FUNCTION_BLOCK Simulation
VAR_INPUT
END_VAR
VAR_OUTPUT
END_VAR
VAR
	tonTaktgeber: ton;	

	xAuslass1: BOOL;	//Es wird Wasser abgelassen
	xAuslass2: BOOL;
	xAuslass3: BOOL;

	uiFuellstandTank1: UINT;	// 0 --> voll; 300 --> leer
	uiFuellstandTank2: UINT;
	uiFuellstandTank3: UINT;	
END_VAR

//Simulation für die Visualisierung
tonTaktgeber(IN:= NOT tonTaktgeber.Q, PT:= T#30MS);

IF tonTaktgeber.Q THEN
	// damit das Simulation mit passabler Geschwindigkeit läuft	

	// Tank leeren
	IF  xAuslass1 THEN
		IF uiFuellstandTank1 < 300 THEN
			uiFuellstandTank1 := uiFuellstandTank1 + 1;
		ELSE
			uiFuellstandTank1 := 300;		
		END_IF
	END_IF

	IF  xAuslass2 THEN
		IF uiFuellstandTank2 < 300 THEN
			uiFuellstandTank2 := uiFuellstandTank2 + 1;
		ELSE
			uiFuellstandTank2 := 300;		
		END_IF
	END_IF

	IF  xAuslass3 THEN
		IF uiFuellstandTank3 < 300 THEN
			uiFuellstandTank3 := uiFuellstandTank3 + 1;
		ELSE
			uiFuellstandTank3 := 300;		
		END_IF
	END_IF
	
	// Tank füllen
	IF DIO.Q1 THEN
		IF uiFuellstandTank1 > 2 THEN
			uiFuellstandTank1 := uiFuellstandTank1 - 2;
		ELSE
			uiFuellstandTank1 := 0;	
		END_IF
	END_IF
	
	IF DIO.Q2 THEN
		IF uiFuellstandTank2 > 2 THEN
			uiFuellstandTank2 := uiFuellstandTank2 - 2;
		ELSE
			uiFuellstandTank2 := 0;	
		END_IF
	END_IF
	
	IF DIO.Q3 THEN
		IF uiFuellstandTank3 > 2 THEN
			uiFuellstandTank3 := uiFuellstandTank3 - 2;
		ELSE
			uiFuellstandTank3 := 0;	
		END_IF
	END_IF
	
END_IF


// Füllstand unten
IF uiFuellstandTank1 > 290 THEN
	VISU.B1 := TRUE;
ELSE
	VISU.B1 := FALSE;
END_IF

IF uiFuellstandTank2 > 290 THEN
	VISU.B3 := TRUE;
ELSE
	VISU.B3 := FALSE;
END_IF

IF uiFuellstandTank3 > 290 THEN
	VISU.B5 := TRUE;
ELSE
	VISU.B5 := FALSE;
END_IF


// Füllstand oben
IF uiFuellstandTank1 < 10 THEN
	VISU.B2 := TRUE;
ELSE
	VISU.B2 := FALSE;
END_IF

IF uiFuellstandTank2 < 10 THEN
	VISU.B4 := TRUE;
ELSE
	VISU.B4 := FALSE;
END_IF

IF uiFuellstandTank3 < 10 THEN
	VISU.B6 := TRUE;
ELSE
	VISU.B6 := FALSE;
END_IF

END_FUNCTION_BLOCK

(* stored: Version 1.1.0.1, ProductVersion 3.1.4022.6
   POU Simulation: Id {54576aa1-06f6-4b89-ab1a-39131b41e0cb}, SpecialFunc None *)
